FUNCTION_BLOCK "FB2017_ZC_M_SINA"
TITLE = FB2017_M_SINA
{ S7_Optimized_Access := 'TRUE' }
AUTHOR : ABH
FAMILY : ZeusControl
VERSION : 1.0
//Bloque de funcion para gestion de dispositivo motor sinamics
   VAR_INPUT
      Pulso1seg { ExternalAccessible := 'False'; ExternalVisible := 'False'; ExternalWritable := 'False'} : Bool;
      Simulacion { ExternalAccessible := 'False'; ExternalVisible := 'False'; ExternalWritable := 'False'} : Bool;
      ACK : Bool;
      SeguridadesOK : Bool;
   END_VAR

   VAR
      HWIDSTW : Array[0.."N_MAX_DISP_M_SINA"] of HW_IO;   // Hardware Identifer set point slot
      HWIDZSW : Array[0.."N_MAX_DISP_M_SINA"] of HW_IO;   // Hardware Identifer actual value slot
      SinaSpeed {InstructionName := 'SinaSpeed'; LibVersion := '1.0'} : Array[0.."N_MAX_DISP_M_SINA"] of SinaSpeed;
   END_VAR

   VAR_TEMP
      for_i : Int;
      for_mux_cambios : Int;
      for_mux : Int;
      t_Activar : Bool;
      t_Frecuencia : Real;
      t_ErrorSinaSpeed : Bool;
      t_ErrorTermico : Bool;
      t_ConfigAxis : Word;
      t_ZSW1 : Bool;
   END_VAR

   VAR CONSTANT
      SOLO_DIRECTO : USInt := 0;
      DIRECTO_INVERSO : USInt := 1;
      TRAZA_DISPOSITIVO : String := 'Dispositivo motor variador ';
      TRAZA_MANUAL : String := ' - En modo manual';
      TRAZA_AUTOMATICO : String := ' - Cambio a modo automatico';
      TRAZA_ACTIVADO : String := '- Activado en modo manual';
      TRAZA_DESACTIVADO : String := '- Desactivado en modo manual';
   END_VAR


BEGIN
	(*
	ZEUS CONTROL, S.A.
	(c)Copyright (2023) All Rights Reserved
	--------------------------------------------------------------------------------------

	Software:       TIA Portal 16
	Restricciones:  PLC serie 1200/1500

	Nombre:         DISPOSITIVO SINAMICS
	Descripcion:    Modelo de dispositivo sinamics (comunicado)

	Dependencias:
	    FC:         FC8_TRAZA_REGISTRO
	    FB:         -
	    DB:         DB2017_DISP_M_SINA
	                DB2018_INST_M_SINA
	                DB1_SYS
	    UDT:        ZC_DISP_M_SINA
	                ZC_MUX

	Change log:

	    Version     Fecha       Tecnico a cargo     Descripcion

	    01.00.00    27.04.2020  (ABH)               Primera version.
	    01.00.01    26.05.2020  (ABH)               Se añade logica como dispositivo motor VF.
	    01.00.02    22.09.2022  (HCR)               Cambio lógica SinaSpeed
	                                                Se añade trazabilidad manualizaciones
	                                                Se añade trazabilidad de activación manual
	    01.00.03    08.11.2022  (HCR)               Cambio lógica enclavamiento
	    01.00.04    18.09.2023  (ABH)               Cambio en tipo de dato de horas de alarma. Se utiliza el tipo de dato ZC_CONTADOR_TIEMPO y el FC15025_ZC_CONTADOR_TIEMPO
	    01.00.05    28.02.2024  (ABH)               Se añade gestion multiplexado para Scada (no indexado)

	//=====================================================================================
	*)

	(* /// <Requires>
(*
UDT: N_MAX_DISP_M_SINA
*)
/// </Requires>

REGION MULTIPLEXADO

	    FOR #for_mux := 0 TO "N_MAX_MUX_DISP" DO

	        IF "DB2017_M_SINA".Mux[#for_mux].Habilitar THEN

	            //  ===========================================================================================================
	            //  Gestionamos solo los tipos
	            IF "DB2017_M_SINA".Mux[#for_mux].Index > 0 THEN

	                /// <Requires>
(*
UDT: N_MAX_DISP_M_SINA
*)
/// </Requires>

REGION LIMITES

	                    //  ===========================================================================================================
	                    //  Limites
	                    IF "DB2017_M_SINA".Mux[#for_mux].Index > "N_MAX_DISP_M_SINA" THEN
	                        "DB2017_M_SINA".Mux[#for_mux].Index := "N_MAX_DISP_M_SINA";
	                    END_IF;
	                    IF "DB2017_M_SINA".Mux[#for_mux].Index >= "N_MAX_DISP_M_SINA" THEN
	                        "DB2017_M_SINA".Mux[#for_mux].MaxVisible := TRUE;
	                    ELSE
	                        "DB2017_M_SINA".Mux[#for_mux].MaxVisible := FALSE;
	                    END_IF;

	                END_REGION


	                /// <Requires>
(*
UDT: N_MAX_DISP_M_SINA
*)
/// </Requires>

REGION CARGA_INICIAL

	                    //  ===========================================================================================================
	                    //  Al detectar un cambio en el indice del dispositivo, cargamos los valores del dispositivo que tenga el indice.
	                    IF "DB2017_M_SINA".Mux[#for_mux].oldIndex <> "DB2017_M_SINA".Mux[#for_mux].Index THEN
	                        "DB2017_M_SINA".Mux[#for_mux].SINA := "DB2017_M_SINA".M_SINA["DB2017_M_SINA".Mux[#for_mux].Index];
	                    END_IF;

	                END_REGION


	                /// <Requires>
(*
UDT: N_MAX_DISP_M_SINA
*)
/// </Requires>

REGION DATOS_LECTURA

	                    //  ===========================================================================================================
	                    //  Movimiento de datos gestionados en FC
	                    "DB2017_M_SINA".Mux[#for_mux].SINA.Hmi_Estado := "DB2017_M_SINA".M_SINA["DB2017_M_SINA".Mux[#for_mux].Index].Hmi_Estado;
	                    IF NOT "DB2017_M_SINA".M_SINA["DB2017_M_SINA".Mux[#for_mux].Index].Estado_AutoMan THEN
	                        "DB2017_M_SINA".Mux[#for_mux].SINA.Orden_ActivarManual := "DB2017_M_SINA".M_SINA["DB2017_M_SINA".Mux[#for_mux].Index].Orden_ActivarManual;
	                    END_IF;
	                    "DB2017_M_SINA".Mux[#for_mux].SINA.Estado_Activado := "DB2017_M_SINA".M_SINA["DB2017_M_SINA".Mux[#for_mux].Index].Estado_Activado;
	                    "DB2017_M_SINA".Mux[#for_mux].SINA.Estado_Enclavado := "DB2017_M_SINA".M_SINA["DB2017_M_SINA".Mux[#for_mux].Index].Estado_Enclavado;
	                    "DB2017_M_SINA".Mux[#for_mux].SINA.Estado_PermisoInvertirSentido := "DB2017_M_SINA".M_SINA["DB2017_M_SINA".Mux[#for_mux].Index].Estado_PermisoInvertirSentido;
	                    "DB2017_M_SINA".Mux[#for_mux].SINA.Estado_RetornoTermico := "DB2017_M_SINA".M_SINA["DB2017_M_SINA".Mux[#for_mux].Index].Estado_RetornoTermico;
	                    "DB2017_M_SINA".Mux[#for_mux].SINA.Estado_EjeBloqueado := "DB2017_M_SINA".M_SINA["DB2017_M_SINA".Mux[#for_mux].Index].Estado_EjeBloqueado;
	                    "DB2017_M_SINA".Mux[#for_mux].SINA.Estado_EjeHabilitado := "DB2017_M_SINA".M_SINA["DB2017_M_SINA".Mux[#for_mux].Index].Estado_EjeHabilitado;
	                    "DB2017_M_SINA".Mux[#for_mux].SINA.Estado_VelocidadLectura := "DB2017_M_SINA".M_SINA["DB2017_M_SINA".Mux[#for_mux].Index].Estado_VelocidadLectura;
	                    "DB2017_M_SINA".Mux[#for_mux].SINA.Estado_VelocidadSalida := "DB2017_M_SINA".M_SINA["DB2017_M_SINA".Mux[#for_mux].Index].Estado_VelocidadSalida;
	                    "DB2017_M_SINA".Mux[#for_mux].SINA.Estado_Estado := "DB2017_M_SINA".M_SINA["DB2017_M_SINA".Mux[#for_mux].Index].Estado_Estado;
	                    "DB2017_M_SINA".Mux[#for_mux].SINA.Estado_CodigoFallo := "DB2017_M_SINA".M_SINA["DB2017_M_SINA".Mux[#for_mux].Index].Estado_CodigoFallo;
	                    "DB2017_M_SINA".Mux[#for_mux].SINA.Alarmas_General := "DB2017_M_SINA".M_SINA["DB2017_M_SINA".Mux[#for_mux].Index].Alarmas_General;
	                    "DB2017_M_SINA".Mux[#for_mux].SINA.Alarmas_Mantenimiento := "DB2017_M_SINA".M_SINA["DB2017_M_SINA".Mux[#for_mux].Index].Alarmas_Mantenimiento;
	                    "DB2017_M_SINA".Mux[#for_mux].SINA.Alarmas_SinaSpeed := "DB2017_M_SINA".M_SINA["DB2017_M_SINA".Mux[#for_mux].Index].Alarmas_SinaSpeed;
	                    "DB2017_M_SINA".Mux[#for_mux].SINA.Alarmas_Termico := "DB2017_M_SINA".M_SINA["DB2017_M_SINA".Mux[#for_mux].Index].Alarmas_Termico;
	                    "DB2017_M_SINA".Mux[#for_mux].SINA.Orden_ActivarAuto := "DB2017_M_SINA".M_SINA["DB2017_M_SINA".Mux[#for_mux].Index].Orden_ActivarAuto;
	                    "DB2017_M_SINA".Mux[#for_mux].SINA.Orden_ConsignaAuto := "DB2017_M_SINA".M_SINA["DB2017_M_SINA".Mux[#for_mux].Index].Orden_ConsignaAuto;
	                    "DB2017_M_SINA".Mux[#for_mux].SINA.Tiempos_Alarma := "DB2017_M_SINA".M_SINA["DB2017_M_SINA".Mux[#for_mux].Index].Tiempos_Alarma;
	                    "DB2017_M_SINA".Mux[#for_mux].SINA.Tiempos_Mantenimiento := "DB2017_M_SINA".M_SINA["DB2017_M_SINA".Mux[#for_mux].Index].Tiempos_Mantenimiento;
	                    "DB2017_M_SINA".Mux[#for_mux].SINA.Aux_oldActivado := "DB2017_M_SINA".M_SINA["DB2017_M_SINA".Mux[#for_mux].Index].Aux_oldActivado;
	                    "DB2017_M_SINA".Mux[#for_mux].SINA.Aux_oldAlarma := "DB2017_M_SINA".M_SINA["DB2017_M_SINA".Mux[#for_mux].Index].Aux_oldAlarma;
	                    "DB2017_M_SINA".Mux[#for_mux].SINA.Aux_oldAutoMan := "DB2017_M_SINA".M_SINA["DB2017_M_SINA".Mux[#for_mux].Index].Aux_oldAutoMan;
	                    "DB2017_M_SINA".Mux[#for_mux].SINA.Config_GrupoAlarma := "DB2017_M_SINA".M_SINA["DB2017_M_SINA".Mux[#for_mux].Index].Config_GrupoAlarma;

	                END_REGION


	                /// <Requires>
(*
UDT: N_MAX_DISP_M_SINA
*)
/// </Requires>

REGION DATOS_ESCRITURA

	                    //  ===========================================================================================================
	                    //  Reinicializamos valor existe cambio
	                    "DB2017_M_SINA".Mux[#for_mux].ExisteCambio := false;

	                    //  ===========================================================================================================
	                    //  Nombre dispositivo
	                    IF "DB2017_M_SINA".Mux[#for_mux].SINA.Hmi_Nombre <> "DB2017_M_SINA".M_SINA["DB2017_M_SINA".Mux[#for_mux].Index].Hmi_Nombre THEN
	                        "DB2017_M_SINA".M_SINA["DB2017_M_SINA".Mux[#for_mux].Index].Hmi_Nombre := "DB2017_M_SINA".Mux[#for_mux].SINA.Hmi_Nombre;
	                        "DB2017_M_SINA".Mux[#for_mux].ExisteCambio := true;
	                    END_IF;

	                    //  ===========================================================================================================
	                    //  Estado auto/manual
	                    IF "DB2017_M_SINA".Mux[#for_mux].SINA.Estado_AutoMan <> "DB2017_M_SINA".M_SINA["DB2017_M_SINA".Mux[#for_mux].Index].Estado_AutoMan THEN
	                        "DB2017_M_SINA".M_SINA["DB2017_M_SINA".Mux[#for_mux].Index].Estado_AutoMan := "DB2017_M_SINA".Mux[#for_mux].SINA.Estado_AutoMan;
	                        "DB2017_M_SINA".Mux[#for_mux].ExisteCambio := true;
	                    END_IF;

	                    //  ===========================================================================================================
	                    //  Ordenes
	                    IF "DB2017_M_SINA".Mux[#for_mux].SINA.Orden_ActivarManual <> "DB2017_M_SINA".M_SINA["DB2017_M_SINA".Mux[#for_mux].Index].Orden_ActivarManual THEN
	                        "DB2017_M_SINA".M_SINA["DB2017_M_SINA".Mux[#for_mux].Index].Orden_ActivarManual := "DB2017_M_SINA".Mux[#for_mux].SINA.Orden_ActivarManual;
	                        "DB2017_M_SINA".Mux[#for_mux].ExisteCambio := true;
	                    END_IF;
	                    IF "DB2017_M_SINA".Mux[#for_mux].SINA.Orden_ResetHoras <> "DB2017_M_SINA".M_SINA["DB2017_M_SINA".Mux[#for_mux].Index].Orden_ResetHoras THEN
	                        "DB2017_M_SINA".M_SINA["DB2017_M_SINA".Mux[#for_mux].Index].Orden_ResetHoras := "DB2017_M_SINA".Mux[#for_mux].SINA.Orden_ResetHoras;
	                        "DB2017_M_SINA".Mux[#for_mux].ExisteCambio := true;
	                    END_IF;
	                    IF "DB2017_M_SINA".Mux[#for_mux].SINA.Orden_ResetFallos <> "DB2017_M_SINA".M_SINA["DB2017_M_SINA".Mux[#for_mux].Index].Orden_ResetFallos THEN
	                        "DB2017_M_SINA".M_SINA["DB2017_M_SINA".Mux[#for_mux].Index].Orden_ResetFallos := "DB2017_M_SINA".Mux[#for_mux].SINA.Orden_ResetFallos;
	                        "DB2017_M_SINA".Mux[#for_mux].ExisteCambio := true;
	                    END_IF;
	                    IF "DB2017_M_SINA".Mux[#for_mux].SINA.Orden_SeleccionInverso <> "DB2017_M_SINA".M_SINA["DB2017_M_SINA".Mux[#for_mux].Index].Orden_SeleccionInverso THEN
	                        "DB2017_M_SINA".M_SINA["DB2017_M_SINA".Mux[#for_mux].Index].Orden_SeleccionInverso := "DB2017_M_SINA".Mux[#for_mux].SINA.Orden_SeleccionInverso;
	                        "DB2017_M_SINA".Mux[#for_mux].ExisteCambio := true;
	                    END_IF;
	                    IF "DB2017_M_SINA".Mux[#for_mux].SINA.Orden_ConsignaManual <> "DB2017_M_SINA".M_SINA["DB2017_M_SINA".Mux[#for_mux].Index].Orden_ConsignaManual THEN
	                        "DB2017_M_SINA".M_SINA["DB2017_M_SINA".Mux[#for_mux].Index].Orden_ConsignaManual := "DB2017_M_SINA".Mux[#for_mux].SINA.Orden_ConsignaManual;
	                        "DB2017_M_SINA".Mux[#for_mux].ExisteCambio := true;
	                    END_IF;

	                    //  ===========================================================================================================
	                    //  Configuracion
	                    IF "DB2017_M_SINA".Mux[#for_mux].SINA.Config_DireccionRetTermicoBit <> "DB2017_M_SINA".M_SINA["DB2017_M_SINA".Mux[#for_mux].Index].Config_DireccionRetTermicoBit THEN
	                        "DB2017_M_SINA".M_SINA["DB2017_M_SINA".Mux[#for_mux].Index].Config_DireccionRetTermicoBit := "DB2017_M_SINA".Mux[#for_mux].SINA.Config_DireccionRetTermicoBit;
	                        "DB2017_M_SINA".Mux[#for_mux].ExisteCambio := true;
	                    END_IF;
	                    IF "DB2017_M_SINA".Mux[#for_mux].SINA.Config_DireccionRetTermicoByte <> "DB2017_M_SINA".M_SINA["DB2017_M_SINA".Mux[#for_mux].Index].Config_DireccionRetTermicoByte THEN
	                        "DB2017_M_SINA".M_SINA["DB2017_M_SINA".Mux[#for_mux].Index].Config_DireccionRetTermicoByte := "DB2017_M_SINA".Mux[#for_mux].SINA.Config_DireccionRetTermicoByte;
	                        "DB2017_M_SINA".Mux[#for_mux].ExisteCambio := true;
	                    END_IF;
	                    IF "DB2017_M_SINA".Mux[#for_mux].SINA.Config_Habilitar <> "DB2017_M_SINA".M_SINA["DB2017_M_SINA".Mux[#for_mux].Index].Config_Habilitar THEN
	                        "DB2017_M_SINA".M_SINA["DB2017_M_SINA".Mux[#for_mux].Index].Config_Habilitar := "DB2017_M_SINA".Mux[#for_mux].SINA.Config_Habilitar;
	                        "DB2017_M_SINA".Mux[#for_mux].ExisteCambio := true;
	                    END_IF;
	                    IF "DB2017_M_SINA".Mux[#for_mux].SINA.Config_HabilitarInvertirTermico <> "DB2017_M_SINA".M_SINA["DB2017_M_SINA".Mux[#for_mux].Index].Config_HabilitarInvertirTermico THEN
	                        "DB2017_M_SINA".M_SINA["DB2017_M_SINA".Mux[#for_mux].Index].Config_HabilitarInvertirTermico := "DB2017_M_SINA".Mux[#for_mux].SINA.Config_HabilitarInvertirTermico;
	                        "DB2017_M_SINA".Mux[#for_mux].ExisteCambio := true;
	                    END_IF;
	                    IF "DB2017_M_SINA".Mux[#for_mux].SINA.Config_HabilitarMantenimiento <> "DB2017_M_SINA".M_SINA["DB2017_M_SINA".Mux[#for_mux].Index].Config_HabilitarMantenimiento THEN
	                        "DB2017_M_SINA".M_SINA["DB2017_M_SINA".Mux[#for_mux].Index].Config_HabilitarMantenimiento := "DB2017_M_SINA".Mux[#for_mux].SINA.Config_HabilitarMantenimiento;
	                        "DB2017_M_SINA".Mux[#for_mux].ExisteCambio := true;
	                    END_IF;
	                    IF "DB2017_M_SINA".Mux[#for_mux].SINA.Config_HabilitarRetornoTermico <> "DB2017_M_SINA".M_SINA["DB2017_M_SINA".Mux[#for_mux].Index].Config_HabilitarRetornoTermico THEN
	                        "DB2017_M_SINA".M_SINA["DB2017_M_SINA".Mux[#for_mux].Index].Config_HabilitarRetornoTermico := "DB2017_M_SINA".Mux[#for_mux].SINA.Config_HabilitarRetornoTermico;
	                        "DB2017_M_SINA".Mux[#for_mux].ExisteCambio := true;
	                    END_IF;
	                    IF "DB2017_M_SINA".Mux[#for_mux].SINA.Config_K_Velocidad <> "DB2017_M_SINA".M_SINA["DB2017_M_SINA".Mux[#for_mux].Index].Config_K_Velocidad THEN
	                        "DB2017_M_SINA".M_SINA["DB2017_M_SINA".Mux[#for_mux].Index].Config_K_Velocidad := "DB2017_M_SINA".Mux[#for_mux].SINA.Config_K_Velocidad;
	                        "DB2017_M_SINA".Mux[#for_mux].ExisteCambio := true;
	                    END_IF;
	                    IF "DB2017_M_SINA".Mux[#for_mux].SINA.Config_VelocidadMax <> "DB2017_M_SINA".M_SINA["DB2017_M_SINA".Mux[#for_mux].Index].Config_VelocidadMax THEN
	                        "DB2017_M_SINA".M_SINA["DB2017_M_SINA".Mux[#for_mux].Index].Config_VelocidadMax := "DB2017_M_SINA".Mux[#for_mux].SINA.Config_VelocidadMax;
	                        "DB2017_M_SINA".Mux[#for_mux].ExisteCambio := true;
	                    END_IF;
	                    IF "DB2017_M_SINA".Mux[#for_mux].SINA.Config_VelocidadMin <> "DB2017_M_SINA".M_SINA["DB2017_M_SINA".Mux[#for_mux].Index].Config_VelocidadMin THEN
	                        "DB2017_M_SINA".M_SINA["DB2017_M_SINA".Mux[#for_mux].Index].Config_VelocidadMin := "DB2017_M_SINA".Mux[#for_mux].SINA.Config_VelocidadMin;
	                        "DB2017_M_SINA".Mux[#for_mux].ExisteCambio := true;
	                    END_IF;


	                    //  ===========================================================================================================
	                    //  Tiempos
	                    IF "DB2017_M_SINA".Mux[#for_mux].SINA.Tiempos_SetPointTiempoAlarma <> "DB2017_M_SINA".M_SINA["DB2017_M_SINA".Mux[#for_mux].Index].Tiempos_SetPointTiempoAlarma THEN
	                        "DB2017_M_SINA".M_SINA["DB2017_M_SINA".Mux[#for_mux].Index].Tiempos_SetPointTiempoAlarma := "DB2017_M_SINA".Mux[#for_mux].SINA.Tiempos_SetPointTiempoAlarma;
	                        "DB2017_M_SINA".Mux[#for_mux].ExisteCambio := true;
	                    END_IF;
	                    IF "DB2017_M_SINA".Mux[#for_mux].SINA.Tiempos_SetPointMantenimiento <> "DB2017_M_SINA".M_SINA["DB2017_M_SINA".Mux[#for_mux].Index].Tiempos_SetPointMantenimiento THEN
	                        "DB2017_M_SINA".M_SINA["DB2017_M_SINA".Mux[#for_mux].Index].Tiempos_SetPointMantenimiento := "DB2017_M_SINA".Mux[#for_mux].SINA.Tiempos_SetPointMantenimiento;
	                        "DB2017_M_SINA".Mux[#for_mux].ExisteCambio := true;
	                    END_IF;

	                END_REGION


	                /// <Requires>
(*
UDT: N_MAX_DISP_M_SINA
*)
/// </Requires>

REGION GESTION_CAMBIOS

	                    //  ===========================================================================================================
	                    //  Si existe cambios en el dispositivo generados por SCADA, actualizamos los datos en el resto de multiplexados,
	                    //  en caso de que este abierto el mismo dispositivo.
	                    IF "DB2017_M_SINA".Mux[#for_mux].ExisteCambio THEN

	                        //  Recorremos todos los multiplexados
	                        FOR #for_mux_cambios := 0 TO "N_MAX_MUX_DISP" DO

	                            //  No miramos el multiplexado actual
	                            IF #for_mux_cambios <> #for_mux THEN

	                                //  En caso de que este seleccionado el mismo indice, movemos el dispositivo al multiplexado
	                                //  correspondiente
	                                IF "DB2017_M_SINA".Mux[#for_mux].Index = "DB2017_M_SINA".Mux[#for_mux_cambios].Index THEN
	                                    "DB2017_M_SINA".Mux[#for_mux_cambios].SINA := "DB2017_M_SINA".M_SINA["DB2017_M_SINA".Mux[#for_mux].Index];
	                                END_IF;

	                            END_IF;

	                        END_FOR;
	                        "DB2017_M_SINA".Mux[#for_mux].ExisteCambio := FALSE;
	                    END_IF;

	                END_REGION

	            END_IF;

	        ELSE

	            "DB2017_M_SINA".Mux[#for_mux].ExisteCambio := FALSE;
	            "DB2017_M_SINA".Mux[#for_mux].Index := 0;

	        END_IF;

	        //  ===========================================================================================================
	        //  Valor anterior del indice
	        "DB2017_M_SINA".Mux[#for_mux].oldIndex := "DB2017_M_SINA".Mux[#for_mux].Index;

	    END_FOR;

	END_REGION


	/// <Requires>
(*
UDT: N_MAX_DISP_M_SINA
*)
/// </Requires>

REGION LOGICA_DEL_DISPOSITIVO

	    // =============================================================================
	    // Resetear todas las alarmas para que se vuelvan a generar
	    FOR #for_i := 0 TO "N_MAX_DISP_AGRUP" DO
	        "DB2017_M_SINA".Agrup[#for_i].AlgunaAlarma := FALSE;
	        "DB2017_M_SINA".Agrup[#for_i].AlgunaEnManual := FALSE;
	    END_FOR;

	    FOR #for_i := 1 TO "N_MAX_DISP_M_SINA" DO

	        /// <Requires>
(*
UDT: N_MAX_DISP_M_SINA
*)
/// </Requires>

REGION LIMITE_GRUPO_ALARMA

	            IF "DB2017_M_SINA".M_SINA[#for_i].Config_GrupoAlarma < 0 THEN
	                "DB2017_M_SINA".M_SINA[#for_i].Config_GrupoAlarma := 0;
	            END_IF;
	            IF "DB2017_M_SINA".M_SINA[#for_i].Config_GrupoAlarma > "N_MAX_DISP_AGRUP" THEN
	                "DB2017_M_SINA".M_SINA[#for_i].Config_GrupoAlarma := "N_MAX_DISP_AGRUP";
	            END_IF;

	        END_REGION

	        // =============================================================================
	        // DISPOSITIVO HABILITADO
	        // =============================================================================
	        IF "DB2017_M_SINA".M_SINA[#for_i].Config_Habilitar THEN

	            // =============================================================================
	            //  PUESTA A CERO DE LA SALIDA
	            #t_Activar := FALSE;
	            #t_Frecuencia := 0.0;

	            // =============================================================================
	            //  INICIALIZACION DE VALORES QUE SIEMPRE TIENEN QUE ESTAR A 1 EN LA PALABRA DE MANDO
	            #t_ConfigAxis := 16#003F;


	            /// <Requires>
(*
UDT: N_MAX_DISP_M_SINA
*)
/// </Requires>

REGION LECTURA_VALORES_DE_LA_TARJETA

	                // =============================================================================
	                // RETORNO TERMICO
	                IF "DB2017_M_SINA".M_SINA[#for_i].Config_DireccionRetTermicoByte >= 0 THEN
	                    "DB2017_M_SINA".M_SINA[#for_i].Estado_RetornoTermico := PEEK_BOOL(area := 16#81,
	                                                                                      dbNumber := 0,
	                                                                                      byteOffset := "DB2017_M_SINA".M_SINA[#for_i].Config_DireccionRetTermicoByte,
	                                                                                      bitOffset := "DB2017_M_SINA".M_SINA[#for_i].Config_DireccionRetTermicoBit);
	                    IF "DB2017_M_SINA".M_SINA[#for_i].Config_HabilitarInvertirTermico THEN
	                        "DB2017_M_SINA".M_SINA[#for_i].Estado_RetornoTermico := NOT (PEEK_BOOL(area := 16#81,
	                                                                                               dbNumber := 0,
	                                                                                               byteOffset := "DB2017_M_SINA".M_SINA[#for_i].Config_DireccionRetTermicoByte,
	                                                                                               bitOffset := "DB2017_M_SINA".M_SINA[#for_i].Config_DireccionRetTermicoBit));
	                    END_IF;
	                END_IF;

	            END_REGION


	            /// <Requires>
(*
UDT: N_MAX_DISP_M_SINA
*)
/// </Requires>

REGION MODOS_DE_TRABAJO

	                // =============================================================================
	                //  RESET CON LOCKOUT
	                IF #SinaSpeed[#for_i].Lockout AND NOT #Simulacion THEN
	                    "DB2017_M_SINA".M_SINA[#for_i].Orden_ActivarManual := FALSE;
	                    "DB2017_M_SINA".M_SINA[#for_i].Orden_ActivarAuto := FALSE;
	                END_IF;

	                // =============================================================================
	                //  MODO MANUAL
	                IF "DB2017_M_SINA".M_SINA[#for_i].Estado_AutoMan THEN
	                    "DB2017_M_SINA".Agrup["DB2017_M_SINA".M_SINA[#for_i].Config_GrupoAlarma].AlgunaEnManual := TRUE;
	                    IF "DB2017_M_SINA".M_SINA[#for_i].Orden_ActivarManual AND NOT "DB2017_M_SINA".M_SINA[#for_i].Estado_Enclavado AND #SeguridadesOK AND NOT "DB2017_M_SINA".M_SINA[#for_i].Alarmas_Termico THEN
	                        #t_Activar := TRUE;
	                        #t_Frecuencia := "DB2017_M_SINA".M_SINA[#for_i].Orden_ConsignaManual;
	                    ELSE
	                        #t_Activar := FALSE;
	                        #t_Frecuencia := 0.0;
	                        "DB2017_M_SINA".M_SINA[#for_i].Orden_ActivarManual := FALSE;
	                    END_IF;
	                ELSE
	                    "DB2017_M_SINA".M_SINA[#for_i].Orden_ActivarManual := FALSE;
	                END_IF;

	                // =============================================================================
	                //  MODO AUTO
	                IF NOT "DB2017_M_SINA".M_SINA[#for_i].Estado_AutoMan THEN
	                    "DB2017_M_SINA".M_SINA[#for_i].Estado_VelocidadSalida := "DB2017_M_SINA".M_SINA[#for_i].Orden_ConsignaAuto;
	                    IF "DB2017_M_SINA".M_SINA[#for_i].Orden_ActivarAuto AND NOT "DB2017_M_SINA".M_SINA[#for_i].Estado_Enclavado AND #SeguridadesOK AND NOT "DB2017_M_SINA".M_SINA[#for_i].Alarmas_Termico THEN
	                        #t_Activar := TRUE;
	                        #t_Frecuencia := "DB2017_M_SINA".M_SINA[#for_i].Orden_ConsignaAuto;
	                    ELSE
	                        #t_Activar := FALSE;
	                        #t_Frecuencia := 0.0;
	                    END_IF;


	                    "DB2017_M_SINA".M_SINA[#for_i].Orden_ActivarManual := "DB2017_M_SINA".M_SINA[#for_i].Estado_Activado;
	                    "DB2017_M_SINA".M_SINA[#for_i].Orden_ConsignaManual := "DB2017_M_SINA".M_SINA[#for_i].Orden_ConsignaAuto;

	                END_IF;

	            END_REGION


	            /// <Requires>
(*
UDT: N_MAX_DISP_M_SINA
*)
/// </Requires>

REGION ESTADO_DEL_DISPOSITIVO

	                // =============================================================================
	                //  MOTOR SIMULADO Y NO SIMULADO
	                IF #Simulacion THEN

	                    IF #t_Activar THEN
	                        "DB2017_M_SINA".M_SINA[#for_i].Estado_Activado := TRUE;
	                    ELSE
	                        "DB2017_M_SINA".M_SINA[#for_i].Estado_Activado := FALSE;
	                    END_IF;

	                    "DB2017_M_SINA".M_SINA[#for_i].Estado_VelocidadLectura := #t_Frecuencia;

	                ELSE
	                    IF "DB2017_M_SINA".M_SINA[#for_i].Estado_EjeHabilitado THEN
	                        "DB2017_M_SINA".M_SINA[#for_i].Estado_Activado := TRUE;
	                    ELSE
	                        "DB2017_M_SINA".M_SINA[#for_i].Estado_Activado := FALSE;
	                    END_IF;

	                    IF #SinaSpeed[#for_i].ActVelocity > 0.0 THEN
	                        "DB2017_M_SINA".M_SINA[#for_i].Estado_VelocidadLectura := #SinaSpeed[#for_i].ActVelocity * "DB2017_M_SINA".M_SINA[#for_i].Config_VelocidadMax / "DB2017_M_SINA".M_SINA[#for_i].Config_K_Velocidad;
	                    ELSE
	                        "DB2017_M_SINA".M_SINA[#for_i].Estado_VelocidadLectura := #SinaSpeed[#for_i].ActVelocity;
	                    END_IF;


	                END_IF;

	            END_REGION


	            /// <Requires>
(*
UDT: N_MAX_DISP_M_SINA
*)
/// </Requires>

REGION ERRORES

	                // =============================================================================
	                //  CHEQUEO RETORNO TERMICO
	                IF NOT #Simulacion AND "DB2017_M_SINA".M_SINA[#for_i].Config_HabilitarRetornoTermico
	                    AND "DB2017_M_SINA".M_SINA[#for_i].Estado_RetornoTermico THEN
	                    #t_ErrorTermico := TRUE;
	                ELSE
	                    #t_ErrorTermico := FALSE;
	                END_IF;


	                // =============================================================================
	                //  CHEQUEO ERROR DESDE EL BLOQUE SINA SPEED
	                IF NOT #Simulacion AND #SinaSpeed[#for_i].Error AND (#SinaSpeed[#for_i].Status <> 16#8402) THEN
	                    #t_ErrorSinaSpeed := TRUE;
	                ELSE
	                    #t_ErrorSinaSpeed := FALSE;
	                END_IF;


	                // =============================================================================
	                //  TEMPORIZADO DE ERRORES
	                IF #t_ErrorSinaSpeed
	                    AND NOT "DB2017_M_SINA".M_SINA[#for_i].Alarmas_SinaSpeed
	                    AND NOT "DB2017_M_SINA".M_SINA[#for_i].Alarmas_Termico
	                THEN
	                    IF NOT #Simulacion AND #Pulso1seg THEN
	                        "DB2017_M_SINA".M_SINA[#for_i].Tiempos_Alarma += 1;
	                    END_IF;
	                ELSE
	                    "DB2017_M_SINA".M_SINA[#for_i].Tiempos_Alarma := 0;
	                END_IF;


	                // =============================================================================
	                //  ERROR TERMICO
	                IF #t_ErrorTermico THEN
	                    "DB2017_M_SINA".M_SINA[#for_i].Alarmas_Termico := TRUE;
	                END_IF;
	                IF NOT #t_ErrorTermico THEN
	                    "DB2017_M_SINA".M_SINA[#for_i].Alarmas_Termico := FALSE;
	                END_IF;

	                // =============================================================================
	                //  ERROR DESDE EL BLOQUE SINA SPEED
	                IF "DB2017_M_SINA".M_SINA[#for_i].Tiempos_Alarma >= "DB2017_M_SINA".M_SINA[#for_i].Tiempos_SetPointTiempoAlarma AND #t_ErrorSinaSpeed THEN
	                    "DB2017_M_SINA".M_SINA[#for_i].Alarmas_SinaSpeed := TRUE;
	                END_IF;
	                IF NOT #t_ErrorSinaSpeed THEN
	                    "DB2017_M_SINA".M_SINA[#for_i].Alarmas_SinaSpeed := FALSE;
	                END_IF;


	                // =============================================================================
	                //  ERROR GLOBAL
	                "DB2017_M_SINA".M_SINA[#for_i].Alarmas_General := "DB2017_M_SINA".M_SINA[#for_i].Alarmas_Termico OR "DB2017_M_SINA".M_SINA[#for_i].Alarmas_SinaSpeed;

	                // =============================================================================
	                //  SI TENEMOS UN ERROR DESACTIVAMOS LA SALIDA
	                IF "DB2017_M_SINA".M_SINA[#for_i].Alarmas_General THEN
	                    "DB2017_M_SINA".Agrup["DB2017_M_SINA".M_SINA[#for_i].Config_GrupoAlarma].AlgunaAlarma := TRUE;
	                    #t_Activar := FALSE;
	                    "DB2017_M_SINA".M_SINA[#for_i].Orden_ActivarManual := FALSE;
	                END_IF;

	            END_REGION


	            /// <Requires>
(*
UDT: N_MAX_DISP_M_SINA
*)
/// </Requires>

REGION DIAGNOSIS

	                //  =============================================================================
	                //  CONTADOR DE HORAS DE FUNCIONAMIENTO
	                IF "DB2017_M_SINA".M_SINA[#for_i].Orden_ResetHoras THEN
	                    "DB2017_M_SINA".M_SINA[#for_i].Orden_ResetHoras := FALSE;
	                END_IF;
	                IF NOT #Simulacion AND #Pulso1seg AND "DB2017_M_SINA".M_SINA[#for_i].Estado_Activado THEN
	                    "DB2017_M_SINA".M_SINA[#for_i].Tiempos_Mantenimiento += 0.00027778;
	                END_IF;
	                //  =============================================================================
	                //  ALARMA HORAS PARA MANTENIMIENTO ALCANZADOS
	                "DB2017_M_SINA".M_SINA[#for_i].Alarmas_Mantenimiento := FALSE;
	                IF "DB2017_M_SINA".M_SINA[#for_i].Config_HabilitarMantenimiento
	                    AND
	                    "DB2017_M_SINA".M_SINA[#for_i].Tiempos_Mantenimiento > "DB2017_M_SINA".M_SINA[#for_i].Tiempos_SetPointMantenimiento
	                THEN
	                    "DB2017_M_SINA".M_SINA[#for_i].Alarmas_Mantenimiento := TRUE;
	                END_IF;

	            END_REGION


	            /// <Requires>
(*
UDT: N_MAX_DISP_M_SINA
*)
/// </Requires>

REGION ESCRITURA_SALIDA


	                "DB2017_M_SINA".M_SINA[#for_i].Estado_VelocidadSalida := #t_Frecuencia;

	                // =============================================================================
	                //  LIMITAR SALIDA A LOS VALORES ESTABLECIDOS EN EL ELEMENTO
	                IF "DB2017_M_SINA".M_SINA[#for_i].Estado_VelocidadSalida > "DB2017_M_SINA".M_SINA[#for_i].Config_VelocidadMax THEN
	                    "DB2017_M_SINA".M_SINA[#for_i].Estado_VelocidadSalida := "DB2017_M_SINA".M_SINA[#for_i].Config_VelocidadMax;
	                END_IF;

	                IF "DB2017_M_SINA".M_SINA[#for_i].Estado_VelocidadSalida < "DB2017_M_SINA".M_SINA[#for_i].Config_VelocidadMin THEN
	                    "DB2017_M_SINA".M_SINA[#for_i].Estado_VelocidadSalida := "DB2017_M_SINA".M_SINA[#for_i].Config_VelocidadMin;
	                END_IF;


	                (*
	                // =============================================================================
	                //  PERMISO PARA INVERTIR EL SENTIDO DE GIRO
	                "DB52_DISP_M_SINA".SINA[#i].Estado_PermisoInvertirSentido := NOT #tempActivar;

	                // =============================================================================
	                //  REINICIALIZO LA PALABRA DE SALIDAS EN CASO DE QUE HAYAMOS INVERTIDO EL SENTIDO DE GIRO
	                IF "DB52_DISP_M_SINA".SINA[#i].Orden_SeleccionInverso THEN
	                    #tempConfigAxis := 16#00FE;
	                END_IF;
	                *)

	                // =============================================================================
	                //  ESCRITURA SALIDA SI NO ESTA LA ORDEN DE ACTIVAR
	                IF NOT #t_Activar THEN
	                    "DB2017_M_SINA".M_SINA[#for_i].Estado_VelocidadSalida := 0.0;
	                END_IF;




	                // =============================================================================
	                //  CONVERSION DE Hz A VALOR EN RPM
	                IF "DB2017_M_SINA".M_SINA[#for_i].Estado_VelocidadSalida > 0.0 THEN
	                    "DB2017_M_SINA".M_SINA[#for_i].Estado_VelocidadSalida := ("DB2017_M_SINA".M_SINA[#for_i].Estado_VelocidadSalida * "DB2017_M_SINA".M_SINA[#for_i].Config_K_Velocidad) / "DB2017_M_SINA".M_SINA[#for_i].Config_VelocidadMax;
	                ELSE
	                    "DB2017_M_SINA".M_SINA[#for_i].Estado_VelocidadSalida := 0.0;
	                END_IF;

	            END_REGION


	            // =============================================================================
	            //  RESET ORDEN ACTIVAR EN AUTO
	            "DB2017_M_SINA".M_SINA[#for_i].Orden_ActivarAuto := FALSE;
	            "DB2017_M_SINA".M_SINA[#for_i].Estado_Enclavado := FALSE;

	            /// <Requires>
(*
UDT: N_MAX_DISP_M_SINA
*)
/// </Requires>

REGION TRAZABILIDAD_MANUALIZACION

	                IF "DB2017_M_SINA".M_SINA[#for_i].Estado_AutoMan AND NOT "DB2017_M_SINA".M_SINA[#for_i].Aux_oldAutoMan THEN
	                    "FC8_ZC_TRAZA_REGISTRO"(FechaHora := "DB1_SYS".FechaHoraActual,
	                                            Registrar := 1,
	                                            Categoria := "TRAZA_CAT_2_MANUALES",
	                                            Id := #for_i,
	                                            User := "DB1_SYS".Usuario.Actual,
	                                            Texto := CONCAT_STRING(IN1 := #TRAZA_DISPOSITIVO, IN2 := "DB2017_M_SINA".M_SINA[#for_i].Hmi_Nombre, IN3 := #TRAZA_MANUAL));
	                END_IF;

	                IF NOT "DB2017_M_SINA".M_SINA[#for_i].Estado_AutoMan AND "DB2017_M_SINA".M_SINA[#for_i].Aux_oldAutoMan THEN
	                    "FC8_ZC_TRAZA_REGISTRO"(FechaHora := "DB1_SYS".FechaHoraActual,
	                                            Registrar := 1,
	                                            Categoria := "TRAZA_CAT_2_MANUALES",
	                                            Id := #for_i,
	                                            User := "DB1_SYS".Usuario.Actual,
	                                            Texto := CONCAT_STRING(IN1 := #TRAZA_DISPOSITIVO, IN2 := "DB2017_M_SINA".M_SINA[#for_i].Hmi_Nombre, IN3 := #TRAZA_AUTOMATICO));
	                END_IF;

	                IF "DB2017_M_SINA".M_SINA[#for_i].Estado_AutoMan AND "DB2017_M_SINA".M_SINA[#for_i].Estado_Activado AND NOT "DB2017_M_SINA".M_SINA[#for_i].Aux_oldActivado THEN
	                    "FC8_ZC_TRAZA_REGISTRO"(FechaHora := "DB1_SYS".FechaHoraActual,
	                                            Registrar := 1,
	                                            Categoria := "TRAZA_CAT_2_MANUALES",
	                                            Id := #for_i,
	                                            User := "DB1_SYS".Usuario.Actual,
	                                            Texto := CONCAT_STRING(IN1 := #TRAZA_DISPOSITIVO, IN2 := "DB2017_M_SINA".M_SINA[#for_i].Hmi_Nombre, IN3 := #TRAZA_ACTIVADO));
	                END_IF;

	                IF "DB2017_M_SINA".M_SINA[#for_i].Estado_AutoMan AND NOT "DB2017_M_SINA".M_SINA[#for_i].Estado_Activado AND "DB2017_M_SINA".M_SINA[#for_i].Aux_oldActivado THEN
	                    "FC8_ZC_TRAZA_REGISTRO"(FechaHora := "DB1_SYS".FechaHoraActual,
	                                            Registrar := 1,
	                                            Categoria := "TRAZA_CAT_2_MANUALES",
	                                            Id := #for_i,
	                                            User := "DB1_SYS".Usuario.Actual,
	                                            Texto := CONCAT_STRING(IN1 := #TRAZA_DISPOSITIVO, IN2 := "DB2017_M_SINA".M_SINA[#for_i].Hmi_Nombre, IN3 := #TRAZA_DESACTIVADO));
	                END_IF;

	            END_REGION

	            // =============================================================================
	            // Estado anterior manual/automatico
	            "DB2017_M_SINA".M_SINA[#for_i].Aux_oldAutoMan := "DB2017_M_SINA".M_SINA[#for_i].Estado_AutoMan;
	            "DB2017_M_SINA".M_SINA[#for_i].Aux_oldActivado := "DB2017_M_SINA".M_SINA[#for_i].Estado_Activado;

	        ELSE

	            // =============================================================================
	            // DISPOSITIVO NO HABILITADO
	            // =============================================================================
	            "DB2017_M_SINA".M_SINA[#for_i].Alarmas_General := FALSE;
	            "DB2017_M_SINA".M_SINA[#for_i].Alarmas_Termico := FALSE;
	            "DB2017_M_SINA".M_SINA[#for_i].Alarmas_Mantenimiento := FALSE;
	            "DB2017_M_SINA".M_SINA[#for_i].Alarmas_SinaSpeed := FALSE;
	            "DB2017_M_SINA".M_SINA[#for_i].Estado_RetornoTermico := FALSE;
	            "DB2017_M_SINA".M_SINA[#for_i].Estado_Enclavado := FALSE;
	            "DB2017_M_SINA".M_SINA[#for_i].Orden_ActivarAuto := FALSE;
	            "DB2017_M_SINA".M_SINA[#for_i].Orden_ActivarManual := FALSE;
	            "DB2017_M_SINA".M_SINA[#for_i].Estado_Activado := FALSE;
	            "DB2017_M_SINA".M_SINA[#for_i].Estado_VelocidadLectura := 0.0;

	        END_IF;


	        /// <Requires>
(*
UDT: N_MAX_DISP_M_SINA
*)
/// </Requires>

REGION GESTION_HMI

	            // =============================================================================
	            //  GESTION BITS PARA VISUALIZACION
	            //  Bit     0   Habilitacion
	            //  Bit     1   ManualAutomatico
	            //  Bit     2   Enclavado
	            //  Bit     3   Activado 1
	            //  Bit     4   Activado 2
	            //  Bit     5   Reserva
	            //  Bit     6   Reserva
	            //  Bit     7   Reserva
	            //  Bit     8   Alarma General
	            //  Bit     9   Alarma 1
	            //  Bit     10  Alarma 2
	            //  Bit     11  Alarma 3
	            //  Bit     12  Alarma 4
	            //  Bit     13  Alarma Mantenimiento
	            //  Bit     14  Reserva
	            //  Bit     15  Reserva
	            "DB2017_M_SINA".M_SINA[#for_i].Hmi_Estado.%X0 := "DB2017_M_SINA".M_SINA[#for_i].Config_Habilitar;
	            "DB2017_M_SINA".M_SINA[#for_i].Hmi_Estado.%X1 := "DB2017_M_SINA".M_SINA[#for_i].Estado_AutoMan;
	            "DB2017_M_SINA".M_SINA[#for_i].Hmi_Estado.%X2 := "DB2017_M_SINA".M_SINA[#for_i].Estado_Enclavado;
	            "DB2017_M_SINA".M_SINA[#for_i].Hmi_Estado.%X3 := "DB2017_M_SINA".M_SINA[#for_i].Estado_Activado;
	            //"DB52_DISP_M_SINA".SINA[#i].HMI_Estado.%X3 := FALSE;
	            //"DB52_DISP_M_SINA".SINA[#i].HMI_Estado.%X4 := FALSE;
	            //"DB52_DISP_M_SINA".SINA[#i].HMI_Estado.%X5 := FALSE;
	            //"DB52_DISP_M_SINA".SINA[#i].HMI_Estado.%X6 := FALSE;
	            //"DB52_DISP_M_SINA".SINA[#i].HMI_Estado.%X7 := FALSE;
	            "DB2017_M_SINA".M_SINA[#for_i].Hmi_Estado.%X8 := "DB2017_M_SINA".M_SINA[#for_i].Alarmas_Termico;
	            "DB2017_M_SINA".M_SINA[#for_i].Hmi_Estado.%X9 := "DB2017_M_SINA".M_SINA[#for_i].Alarmas_SinaSpeed;
	            //"DB52_DISP_M_SINA".SINA[#i].HMI_Estado.%X10 := FALSE;
	            //"DB52_DISP_M_SINA".SINA[#i].HMI_Estado.%X11 := FALSE;
	            //"DB52_DISP_M_SINA".SINA[#i].HMI_Estado.%X12 := FALSE;
	            "DB2017_M_SINA".M_SINA[#for_i].Hmi_Estado.%X13 := "DB2017_M_SINA".M_SINA[#for_i].Alarmas_Mantenimiento;
	            //"DB52_DISP_M_SINA".SINA[#i].HMI_Estado.%X14 := FALSE;
	            //"DB52_DISP_M_SINA".SINA[#i].HMI_Estado.%X15 := FALSE;

	        END_REGION


	        /// <Requires>
(*
UDT: N_MAX_DISP_M_SINA
*)
/// </Requires>

REGION GESTION_NUEVA_ALARMA

	            // =============================================================================
	            //  DETECCION DE NUEVA ALARMA
	            IF "DB2017_M_SINA".M_SINA[#for_i].Alarmas_General AND NOT "DB2017_M_SINA".M_SINA[#for_i].Aux_oldAlarma THEN
	                "DB2017_M_SINA".Agrup["DB2017_M_SINA".M_SINA[#for_i].Config_GrupoAlarma].NuevaAlarma := TRUE;
	            END_IF;

	            //  Estado anterior de las alarmas
	            "DB2017_M_SINA".M_SINA[#for_i].Aux_oldAlarma := "DB2017_M_SINA".M_SINA[#for_i].Alarmas_General;

	        END_REGION


	        /// <Requires>
(*
UDT: N_MAX_DISP_M_SINA
*)
/// </Requires>

REGION SINASPEED


	            IF #HWIDSTW[#for_i] <> 0 AND #HWIDZSW[#for_i] <> 0 THEN
	                #SinaSpeed[#for_i](EnableAxis := #t_Activar,
	                                   AckError := "DB2017_M_SINA".M_SINA[#for_i].Orden_ResetFallos OR #ACK,
	                                   SpeedSp := "DB2017_M_SINA".M_SINA[#for_i].Estado_VelocidadSalida,
	                                   RefSpeed := "DB2017_M_SINA".M_SINA[#for_i].Config_K_Velocidad,
	                                   ConfigAxis := #t_ConfigAxis,
	                                   HWIDSTW := #HWIDSTW[#for_i],
	                                   HWIDZSW := #HWIDZSW[#for_i],
	                                   AxisEnabled => "DB2017_M_SINA".M_SINA[#for_i].Estado_EjeHabilitado,
	                                   Lockout => "DB2017_M_SINA".M_SINA[#for_i].Estado_EjeBloqueado,
	                                   Status => "DB2017_M_SINA".M_SINA[#for_i].Estado_Estado,
	                                   DiagId => "DB2017_M_SINA".M_SINA[#for_i].Estado_CodigoFallo);
	            END_IF;

	            // =============================================================================
	            //  ESCRITURA RESET FALLOS
	            IF "DB2017_M_SINA".M_SINA[#for_i].Orden_ResetFallos AND #Pulso1seg THEN  //  Reset de este BIT cada segundo (es suficiente para resetear el Variador)
	                "DB2017_M_SINA".M_SINA[#for_i].Orden_ResetFallos := FALSE;
	            END_IF;

	        END_REGION

	    END_FOR;


	    // =============================================================================
	    //  ACUSE DE NUEVAS ALARMAS
	    IF #ACK THEN
	        FOR #for_i := 0 TO "N_MAX_DISP_AGRUP" DO
	            "DB2017_M_SINA".Agrup["DB2017_M_SINA".M_SINA[#for_i].Config_GrupoAlarma].NuevaAlarma := FALSE;
	        END_FOR;
	    END_IF;


	END_/// <Requires>
(*
UDT: N_MAX_DISP_M_SINA
*)
/// </Requires>

REGION *)


END_FUNCTION_BLOCK

